FUNCTION_BLOCK FB_OnAndOffButtons
VAR_INPUT
	bIsButtonOn : BOOL;
	bIsButtonOff : BOOL;
END_VAR
VAR_OUTPUT
	bLightOfOnAndOffButton : BOOL;
END_VAR
VAR
	fbOn_RTRIG : R_TRIG;
	fbOff_RTRIG : R_TRIG;
END_VAR

// One button turns the light on, the other turns it off
IF bIsButtonOn THEN
	bLightOfOnAndOffButton := TRUE;
	bIsButtonOff := FALSE;
END_IF

IF bIsButtonOff THEN
	bLightOfOnAndOffButton := FALSE;
	bIsButtonOn := FALSE;
END_IF

// Solution using triggers:
//fbOn_RTRIG(clk := bIsButtonOn);
//IF fbOn_RTRIG.Q THEN
//	bLightOfOnAndOffButton := TRUE;
//	fbOn_RTRIG(clk := FALSE);
//END_IF

//fbOff_RTRIG(clk := bIsButtonOff);
//IF fbOff_RTRIG.Q THEN
//	bLightOfOnAndOffButton := FALSE;
//	fbOff_RTRIG(clk := FALSE);
//END_IF

END_FUNCTION_BLOCK

(* stored: Version 1.1.0.1, ProductVersion 3.1.4024.12
   POU FB_OnAndOffButtons: Id {93fa715c-cb09-4f2b-8ea8-c58272dd4677}, SpecialFunc None *)
